FUNCTION_BLOCK FB_CarGroup EXTENDS FB_LinkedList_Master IMPLEMENTS ITF_Car
VAR_INPUT
END_VAR
VAR_OUTPUT
END_VAR
VAR
END_VAR

{attribute 'monitoring' := 'call'}
PROPERTY p_Locked : BOOL
GET
VAR
	i:		UINT;
	itfCar:	ITF_Car;
END_VAR
p_Locked := TRUE;

FOR i := 0 TO ListLength DO
	IF __QUERYINTERFACE( mListGetNode(i), itfCar) THEN
		p_Locked R= NOT itfCar.p_Locked;
	END_IF
END_FOR
END_GET
SET
VAR
	i:		UINT;
	itfCar:	ITF_Car;
END_VAR
FOR i := 0 TO ListLength DO
	IF __QUERYINTERFACE( mListGetNode(i), itfCar) THEN
		itfCar.p_Locked := p_Locked;
	END_IF
END_FOR
END_SET
END_PROPERTY

END_FUNCTION_BLOCK

(* stored: Version 1.1.0.1, ProductVersion 3.1.4024.12
   POU FB_CarGroup: Id {dee57356-43af-4a4c-9e1d-d5468a41ae59}, SpecialFunc None
   Property p_Locked: Id {5d545e78-0a37-4b95-a748-b38f659c9a05}
   Get Get: Id {3782913b-1a3c-49c9-9526-5922edfe5232}
   Set Set: Id {d7c7424c-d126-4d65-8cc0-f4c3b2836cd6} *)
